TYPE ST_PullCharmber :
STRUCT
END_STRUCT
END_TYPE

(* stored: Version 1.1.0.1, ProductVersion 3.1.4024.12
   DUT ST_PullCharmber: Id {35b3a947-9936-4dc6-8bd8-1d63007c6514} *)
